PROGRAM Axis02_Status
VAR
	Always_ON	:	BOOL	:=TRUE	;//상시 ON 
	Always_OFF	:	BOOL	:=FALSE	;//상시 OFF
END_VAR

// NETWORK 1

END_PROGRAM

(* stored: Version 1.1.0.1, ProductVersion 3.1.4024.15
   POU Axis02_Status: Id {6c8f84cb-e148-4c91-9c9e-c81eb8526fa8}, SpecialFunc None *)
